TYPE ST_SafeMovements :
STRUCT

	JogTimer 			:TON;
	JogTrig				 :R_TRIG;
	Jog					:BOOL;
	Conflict				:BOOL;
	ConflictReported		:BOOL;
	ConflictTrig 			:R_TRIG;
	ConflictMessage		:STRING[1024];
	UdID				:UDINT;

END_STRUCT
END_TYPE

(* stored: Version 1.1.0.1, ProductVersion 3.1.4024.11
   DUT ST_SafeMovements: Id {8509bdad-05f7-4cee-af03-a021b253aa7f} *)
